# B&R Automation Studio project lab1_SoftwareOFRobotics
Automation Studio 4.5.2.102

## Configuration Config1

CPU 4PP065.0571-P74, AutomationRuntime D4.52, Build 4.1.2, Vc V4.52.0

### Task classes (Cpu.sw)
```
Cyclic#1:
  Program <- Program.prg
Libraries: Library
```

### Hardware
```
4PP065_0571_P74 : 4PP065.0571-P74 v1.1.2.0
  Connector IF4:
    InternetAddress = 10.0.1.10
    SubnetMask = 255.255.255.0
  Connector IF5:
    ActivateDevice = 1
    Mode = Manual
  ConfigurationID = labBR
  Simulation = 1
```

- Physical/Config1/4PP065_0571_P74/IoMap.iom: same as Physical/Config1/4PP065_0571_P74/Cpu.per
- Physical/Config1/4PP065_0571_P74/PvMap.vvm: same as Physical/Config1/4PP065_0571_P74/Cpu.per
## Logical view

Binary libraries used (declarations not repeated): operator, runtime, astime, AsIecCon

### Package Logical/Libraries - Global libraries

### Library Logical/Libraries/Library (ANSIC)

#### Constants.var - Exported constants
```iecst
VAR CONSTANT
	d_t : REAL := 0.01;
END_VAR
```

#### Library.fun - Exported functions and function blocks
```iecst
{REDUND_ERROR} FUNCTION_BLOCK FB_motor (*TODO: I don't know what this shit do)*) (*$GROUP=User,$CAT=User,$GROUPICON=User.png,$CATICON=User.png*)
	VAR_INPUT
		u_in : {REDUND_UNREPLICABLE} REAL;
		dt : REAL;
	END_VAR
	VAR_OUTPUT
		W : {REDUND_UNREPLICABLE} REAL;
		phi : {REDUND_UNREPLICABLE} REAL;
	END_VAR
	VAR
		Tm : {REDUND_UNREPLICABLE} REAL;
		ke : {REDUND_UNREPLICABLE} REAL;
		Integrator : {REDUND_UNREPLICABLE} FB_Integrator;
	END_VAR
END_FUNCTION_BLOCK

FUNCTION_BLOCK FB_Integrator
	VAR_INPUT
		in : REAL;
		dt : REAL;
	END_VAR
	VAR_OUTPUT
		out : REAL;
	END_VAR
	VAR
		prev_value : REAL;
	END_VAR
END_FUNCTION_BLOCK

FUNCTION_BLOCK FB_Controller
	VAR_INPUT
		e : {REDUND_UNREPLICABLE} REAL;
		dt : REAL;
	END_VAR
	VAR_OUTPUT
		u : {REDUND_UNREPLICABLE} REAL;
	END_VAR
	VAR
		last_sum : REAL;
		sum : REAL;
		a : REAL;
		k_p : REAL;
		k_i : REAL;
		max_abs_value : REAL;
		Integrator : FB_Integrator;
		iyOld : REAL;
	END_VAR
END_FUNCTION_BLOCK
```

#### FB_motor.c
```c
#include <bur/plctypes.h>
#ifdef __cplusplus
	extern "C"
	{
#endif
	#include "Library.h"
#ifdef __cplusplus
	};
#endif
/* TODO: I don't know what this shit do) */
void FB_motor(struct FB_motor* inst)
{
	REAL a = inst->u_in / inst->ke - inst->W;
	REAL b = a / inst->Tm;

	inst->Integrator.in = b;
	FB_Integrator(&inst->Integrator);
	inst->W = inst->Integrator.out;
/*
	inst->Integrator.in = inst->W;
	FB_Integrator(&inst->Integrator);
	inst->phi = inst->Integrator.out;
*/
}
```

#### FB_Integrator.c
```c
#include <bur/plctypes.h>
#ifdef __cplusplus
	extern "C"
	{
#endif
	#include "Library.h"
#ifdef __cplusplus
	};
#endif
/* TODO: Add your comment here */
void FB_Integrator(struct FB_Integrator* inst)
{
	inst->dt = d_t;
	inst->out = d_t* inst->in + inst->prev_value;
	inst->prev_value = inst->out;
}
```

#### FB_Controller.c
```c
#include <bur/plctypes.h>
#ifdef __cplusplus
	extern "C"
	{
#endif
	#include "Library.h"
#ifdef __cplusplus
	};
#endif
/* TODO: Add your comment here */
void FB_Controller(struct FB_Controller* inst)
{
	REAL a = inst->e * inst->k_p;
	REAL b = inst->e * inst->k_i;

//	a = a > inst->max_abs_value ? inst->max_abs_value:a;
//	a = a < inst->max_abs_value ? - inst->max_abs_value : a;

	// Блок ограничения напряжения
	if ( abs(a) < inst->max_abs_value )
	{
		a = a;
	}
	else
	{
		if (a<0)
		{
			a = (-1)* inst->max_abs_value;
		}
		else
		{
			a = inst->max_abs_value;
		}
	}

	inst->Integrator.in = b + inst->iyOld;
	FB_Integrator(&inst->Integrator);

	REAL sum = a + inst->Integrator.out;

	inst->u = sum;

	inst->u = inst->u > inst->max_abs_value ? inst->max_abs_value : inst->u;
	inst->u = inst->u < - inst->max_abs_value ? -inst->max_abs_value: inst->u;

	inst->iyOld = inst->u - sum;

}
```

### Program Logical/Program (ANSIC)

#### Main.c - Init, cyclic, exit code
```c
#include <bur/plctypes.h>

#ifdef _DEFAULT_INCLUDES
	#include <AsDefault.h>
#endif

void _INIT ProgramInit(void)
{
	fb_motor1.ke = 0.15;
	fb_motor1.Tm = 0.3;
	fb_motor1.u_in = 0;
	fb_motor1.dt = 0.001;

	fb_motor2.ke = 0.15;
	fb_motor2.Tm = 0.3;
	fb_motor2.u_in = 0;
	fb_motor2.dt = 0.001;

	fb_controller.k_p = 0.45;
	fb_controller.k_i = 1.5;
	fb_controller.max_abs_value = 25.0;
	fb_controller.dt = 0.001;

	speed = 0;
	speed2 = 0;
	counter = 0;
	enable = 1;
}

void _CYCLIC ProgramCyclic(void)
{
	if (enable)
	{
		if (counter == 300)
		{
			speed = 0;
			speed2 = 0;
			counter = 0;
		}
		else if (counter == 100){
			speed = 50;
			speed2 = 50;
		}
		fb_controller.e = speed - fb_motor1.W;
		FB_Controller(&fb_controller);

		fb_motor1.u_in = fb_controller.u;
		FB_motor(&fb_motor1);

		fb_motor2.u_in = speed2 * fb_motor2.ke;
		FB_motor(&fb_motor2);

		counter++;
	}
}

void _EXIT ProgramExit(void)
{

}
```

#### Variables.var - Local variables
```iecst
VAR
	speed2 : REAL;
	fb_controller : FB_Controller;
	fb_motor1 : FB_motor;
	fb_motor2 : FB_motor;
	counter : UINT;
	speed : REAL;
	enable : BOOL;
END_VAR
```
